// SIMATIC S7-200 SMART project (STEP 7-Micro/WIN SMART), CPU SR40

SYMBOL_TABLE 系统符号
Always_On        SM0.0    // 始终接通
First_Scan_On    SM0.1    // 仅在第一个扫描周期时接通
END_SYMBOL_TABLE

ORGANIZATION_BLOCK MAIN:OB1
TITLE=程序注释
BEGIN
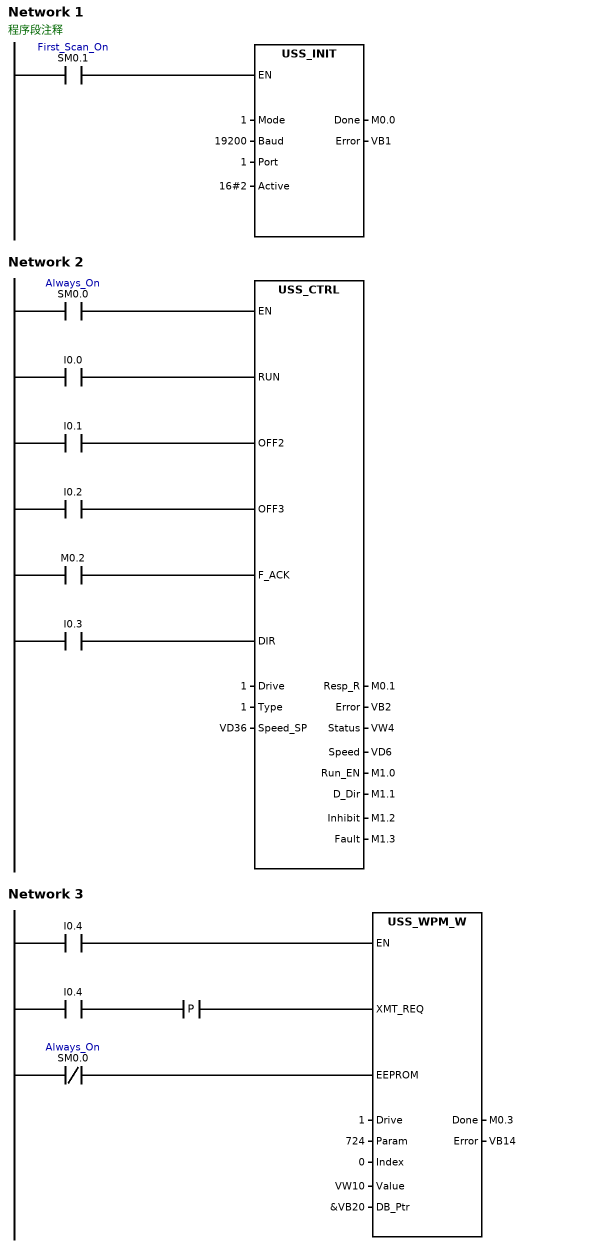
Network 1
// 程序段注释
LD     First_Scan_On:SM0.1
CALL   USS_INIT:SBR2, 1, 19200, 1, 16#2, M0.0, VB1
Network 2
LD     Always_On:SM0.0
=      L60.0
LD     I0.0
=      L63.7
LD     I0.1
=      L63.6
LD     I0.2
=      L63.5
LD     M0.2
=      L63.4
LD     I0.3
=      L63.3
LD     L60.0
CALL   USS_CTRL:SBR5, L63.7, L63.6, L63.5, L63.4, L63.3, 1, 1, VD36, M0.1, VB2, VW4, VD6, M1.0, M1.1, M1.2, M1.3
Network 3
LD     I0.4
=      L60.0
LD     I0.4
EU
=      L63.7
LDN    Always_On:SM0.0
=      L63.6
LD     L60.0
CALL   USS_WPM_W:SBR11, L63.7, L63.6, 1, 724, 0, VW10, &VB20, M0.3, VB14
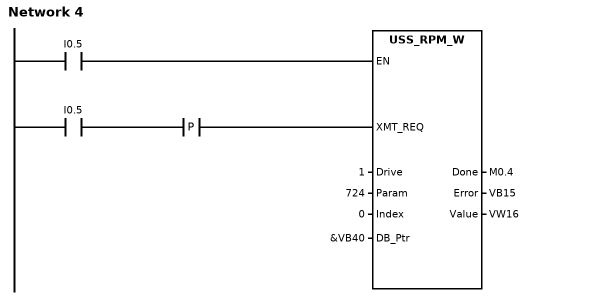
Network 4
LD     I0.5
=      L60.0
LD     I0.5
EU
=      L63.7
LD     L60.0
CALL   USS_RPM_W:SBR12, L63.7, 1, 724, 0, &VB40, M0.4, VB15, VW16
END_ORGANIZATION_BLOCK

// SBR1: protected block, not included

// SBR2: protected block, not included

// SBR3: protected block, not included

// SBR4: protected block, not included

// SBR5: protected block, not included

// SBR6: protected block, not included

// SBR7: protected block, not included

// SBR8: protected block, not included

// SBR9: protected block, not included

// SBR10: protected block, not included

// SBR11: protected block, not included
